(* IEC 61131-3 sources: PLC_1/exp_2/build, 2 files *)

(* ---- plc.st ---- *)
TYPE
  LOGLEVEL : (CRITICAL, WARNING, INFO, DEBUG) := INFO;
END_TYPE

FUNCTION_BLOCK LOGGER
  VAR_INPUT
    TRIG : BOOL;
    MSG : STRING;
    LEVEL : LOGLEVEL := INFO;
  END_VAR
  VAR
    TRIG0 : BOOL;
  END_VAR

  IF TRIG AND NOT TRIG0 THEN
  {{
   LogMessage(GetFbVar(LEVEL),(char*)GetFbVar(MSG, .body),GetFbVar(MSG, .len));
  }}
  END_IF;
  TRIG0:=TRIG;
END_FUNCTION_BLOCK

PROGRAM exp2
  VAR_INPUT
    Start : BOOL;
    Stop : BOOL;
  END_VAR
  VAR_OUTPUT
    Motor : BOOL;
  END_VAR

  Motor := NOT(Stop) AND Start;
END_PROGRAM

CONFIGURATION Config0

  RESOURCE Res0 ON PLC
    TASK task0(INTERVAL := T#20ms,PRIORITY := 0);
    PROGRAM instance0 WITH task0 : exp2;
  END_RESOURCE
END_CONFIGURATION

(* ---- generated_plc.st ---- *)
PROGRAM exp2
  VAR_INPUT
    Start : BOOL;
    Stop : BOOL;
  END_VAR
  VAR_OUTPUT
    Motor : BOOL;
  END_VAR

  Motor := NOT(Stop) AND Start;
END_PROGRAM

CONFIGURATION Config0

  RESOURCE Res0 ON PLC
    TASK task0(INTERVAL := T#20ms,PRIORITY := 0);
    PROGRAM instance0 WITH task0 : exp2;
  END_RESOURCE
END_CONFIGURATION
